PROGRAM Scaling_And_Conversions
VAR
	Rotor_Actual_Torque_Scaled : REAL;
	Feedroll_Actual_Torque_Scaled : REAL;
	
	Rotor_Actual_Current_Scaled : REAL;
	Feedroll_Actual_Current_Scaled : REAL;
	
	Rotor_DC_Bus_Voltage_Scaled : REAL;
	Feedroll_DC_Bus_Voltage_Scaled : REAL;
END_VAR

Rotor_Actual_Torque_Scaled := INT_TO_REAL(GVL_Pelletizer.MyPelletizer.Rotor_VFD.VFD_Actual_Torque) / 10;
Feedroll_Actual_Torque_Scaled := INT_TO_REAL(GVL_Pelletizer.MyPelletizer.Feedroll_VFD.VFD_Actual_Torque) / 10;

Rotor_Actual_Current_Scaled := INT_TO_REAL(GVL_Pelletizer.MyPelletizer.Rotor_VFD.VFD_Actual_Current) / 10;
Feedroll_Actual_Current_Scaled := INT_TO_REAL(GVL_Pelletizer.MyPelletizer.Feedroll_VFD.VFD_Actual_Current) / 10;

Rotor_DC_Bus_Voltage_Scaled := UDINT_TO_REAL(GVL_Pelletizer.MyPelletizer.Rotor_VFD.VFD_DC_Bus_Voltage) / 1000;
Feedroll_DC_Bus_Voltage_Scaled := UDINT_TO_REAL(GVL_Pelletizer.MyPelletizer.Feedroll_VFD.VFD_DC_Bus_Voltage) / 1000;

END_PROGRAM

(* stored: Version 1.1.0.1, ProductVersion 3.1.4024.12
   POU Scaling_And_Conversions: Id {8e970592-64c0-43ad-8110-566d9f1a776b}, SpecialFunc None *)
